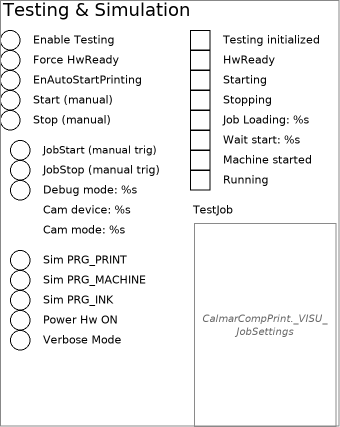
VISUALIZATION _VISU_PrgPrint_test  // 340x427
VAR_IN_OUT
	mInst : FB_PrgPrint_test;
END_VAR
    Ellipse (0,30 20x20)
        toggle mInst._bEnTesting
    Rectangle (30,30 120x20), "Enable Testing"
    Ellipse (0,70 20x20)
        toggle mInst._bEnAutoStartPrinting
    Rectangle (30,70 120x20), "EnAutoStartPrinting"
    Ellipse (10,180 20x20)
        toggle mInst._bEnVerboseMode
    Rectangle (40,180 120x20), "Debug mode: %s", text variable: mInst._eLogLevel
    Ellipse (10,270 20x20)
        toggle mInst._bSimPrgMachine
    Rectangle (40,270 120x20), "Sim PRG_MACHINE"
    Ellipse (10,290 20x20)
        toggle mInst._bSimPrgInk
    Rectangle (40,290 120x20), "Sim PRG_INK"
    Ellipse (10,250 20x20)
        toggle mInst._bSimPrgPrint
    Rectangle (40,250 120x20), "Sim PRG_PRINT"
    RoundedRectangle (190,30 20x20), colour toggle: mInst.bInitialized
    Rectangle (220,30 120x20), "Testing initialized"
    RoundedRectangle (190,50 20x20), tooltip "All enabled CBs are in OP", colour toggle: mInst.bHwReady
    Rectangle (220,50 120x20), "HwReady"
    RoundedRectangle (190,70 20x20), colour toggle: mInst.bStarting
    Rectangle (220,70 120x20), "Starting"
    RoundedRectangle (190,90 20x20), colour toggle: mInst.bStopping
    Rectangle (220,90 120x20), "Stopping"
    RoundedRectangle (190,170 20x20), colour toggle: mInst.bRunning
    Rectangle (220,170 120x20), "Running"
    Rectangle (220,110 120x20), "Job Loading: %s", tooltip "Timeout after: %s", text variable: mInst.LoadTestJob.tExecute.ET
        p4168582468: mInst.LoadTestJob.tExecute.PT
    RoundedRectangle (190,110 20x20), colour toggle: mInst.LoadTestJob.bbusy
    Rectangle (220,130 120x20), "Wait start: %s", text variable: mInst.TestStartSequence.tWaitJobStart.ET
    RoundedRectangle (190,130 20x20), colour toggle: mInst.TestStartSequence.tWaitJobStart.IN
    Rectangle (40,200 120x20), "Cam device: %s", text variable: mInst.eCameraDevice
        OnMouseClick: write the text variable via Default
    Rectangle (40,220 120x20), "Cam mode: %s", text variable: mInst.eCameraMode
        OnMouseClick: write the text variable via Default
    Ellipse (0,90 20x20)
        toggle mInst.bStart
    Rectangle (30,90 120x20), "Start (manual)"
    Ellipse (0,110 20x20)
        toggle mInst.bStop
    Rectangle (30,110 120x20), "Stop (manual)"
    Rectangle (0,0 200x20), "Testing & Simulation"
    Ellipse (10,140 20x20)
        tap mInst._pAdsPu^.sI_Start.bI_Command
        toggle mInst.bStart
    Rectangle (40,140 120x20), "JobStart (manual trig)"
    Ellipse (10,160 20x20)
        tap mInst._pAdsPu^.sI_Stop.bI_Command
        toggle mInst.bStop
    Rectangle (40,160 120x20), "JobStop (manual trig)"
    Frame (194,223 142x204)
        shows CalmarCompPrint._VISU_JobSettings(mInst := mInst.sJobConfig)
    RoundedRectangle (190,150 20x20), colour toggle: mInst.bRunMachine
    Rectangle (220,150 120x20), "Machine started"
    Rectangle (190,200 120x20), "TestJob"
    Ellipse (0,50 20x20)
        toggle mInst._bForceHwReady
    Rectangle (30,50 120x20), "Force HwReady"
    Ellipse (10,310 20x20)
        toggle mInst.bO_Power24V_ON
    Rectangle (40,310 120x20), "Power Hw ON"
    Ellipse (10,330 20x20)
        toggle mInst._bEnVerboseMode
    Rectangle (40,330 120x20), "Verbose Mode"
END_VISUALIZATION

(* stored: Version 1.1.0.1, ProductVersion 3.1.4024.11
   Visu _VISU_PrgPrint_test: Id {4477f59f-af0d-488f-8f11-0bc7d5f0922f} *)
